FUNCTION_BLOCK MovingStatusType2 (* Protection layer *)
  (* Standard: 61499-2 *)
  (* Version 1.0, 2011-04-20, Sandeep Patil, The University of Auckland, First build. *)
  PACKAGE Main;
  (* Compiler header: package fb.rt.pnp; *)
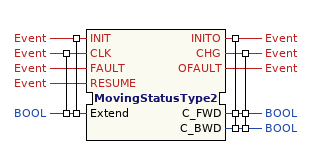
  EVENT_INPUT
    INIT WITH Extend; (* Initialization Request *)
    CLK WITH Extend; (* Clock signal *)
    FAULT;
    RESUME;
  END_EVENT
  EVENT_OUTPUT
    INITO WITH C_FWD, C_BWD; (* Initialization Confirm *)
    CHG WITH C_FWD, C_BWD; (* Data outputs changed *)
    OFAULT;
  END_EVENT
  VAR_INPUT
    Extend : BOOL; (* Move forwards *)
  END_VAR
  VAR_OUTPUT
    C_FWD : BOOL; (* Confirmed move forwards *)
    C_BWD : BOOL; (* Confirmed move backwards *)
  END_VAR
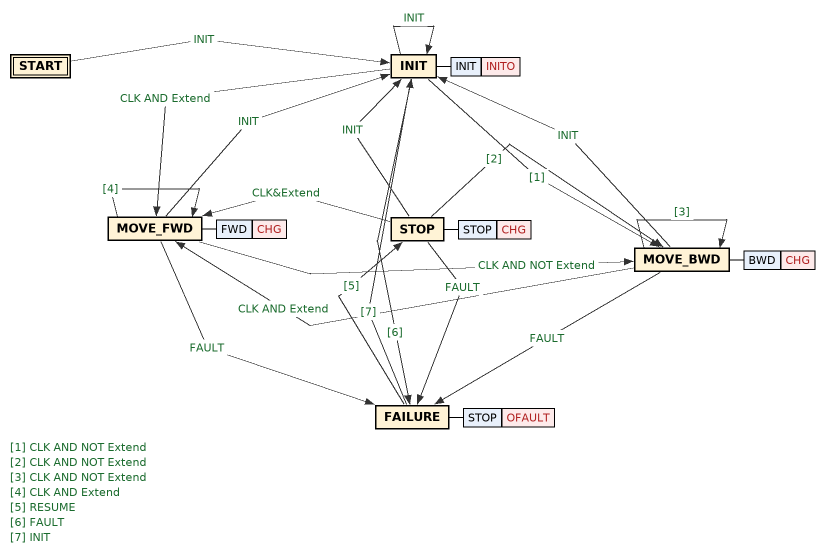
  EC_STATES
    START; (* Initial State *)
    INIT : INIT -> INITO; (* Initialization *)
    MOVE_FWD : FWD -> CHG;
    MOVE_BWD : BWD -> CHG;
    STOP : STOP -> CHG;
    FAILURE : STOP -> OFAULT;
  END_STATES
  EC_TRANSITIONS
    START TO INIT := INIT;
    INIT TO MOVE_FWD := CLK AND Extend;
    INIT TO MOVE_BWD := CLK AND NOT Extend;
    MOVE_FWD TO FAILURE := FAULT;
    STOP TO FAILURE := FAULT;
    MOVE_BWD TO FAILURE := FAULT;
    STOP TO MOVE_FWD := CLK&Extend;
    STOP TO MOVE_BWD := CLK AND NOT Extend;
    FAILURE TO STOP := RESUME;
    MOVE_FWD TO MOVE_BWD := CLK AND NOT Extend;
    MOVE_BWD TO MOVE_FWD := CLK AND Extend;
    MOVE_FWD TO MOVE_FWD := CLK AND Extend;
    MOVE_BWD TO MOVE_BWD := CLK AND NOT Extend;
    INIT TO FAILURE := FAULT;
    MOVE_FWD TO INIT := INIT;
    STOP TO INIT := INIT;
    MOVE_BWD TO INIT := INIT;
    FAILURE TO INIT := INIT;
    INIT TO INIT := INIT;
  END_TRANSITIONS
  ALGORITHM INIT IN ST: (* Initialization algorithm *)
INIT:=FALSE;
C_FWD := FALSE;
C_BWD := FALSE;
  END_ALGORITHM
  ALGORITHM FWD IN ST: (* Normally executed algorithm *)
C_FWD := TRUE;
C_BWD := FALSE;
  END_ALGORITHM
  ALGORITHM BWD IN ST:
C_FWD := FALSE;
C_BWD := TRUE;
  END_ALGORITHM
  ALGORITHM STOP IN ST:
C_FWD := FALSE;
C_BWD := FALSE;
  END_ALGORITHM
END_FUNCTION_BLOCK
